FUNCTION_BLOCK GearSequenceGoHome EXTENDS GearSequence IMPLEMENTS ZCore.ISequence
VAR
  _step : ZCore.Step(GearStep.GohomeBegin, GearStep.GohomeEnd);
  _timer : ZAux.Timer;
END_VAR

IF NOT Busy THEN
  RETURN;
END_IF

IF OnStart(_step) THEN
  ; // init custom sequence variables here ...
END_IF

IF OnStop() THEN
  RETURN; // external stop was triggered
END_IF

IF OnHalt() THEN
  ; // Halting := TRUE; // Uncomment to acknowledge that the sequence is halting
END_IF

REPEAT
  LogStep();

  CASE _step.Index OF
    (* -------------------------------------------------------------------------------------------------------------------------------- *)
    GearStep.GoHomeBegin:
    (* -------------------------------------------------------------------------------------------------------------------------------- *)

      _step.SetNext(index:=GearStep.GoHomePositionX);

	(* -------------------------------------------------------------------------------------------------------------------------------- *)
    GearStep.GoHomePositionX:
    (* -------------------------------------------------------------------------------------------------------------------------------- *)
      IF _step.OnEntry()
      THEN        
        _axis.PositionX.MoveAbsoluteAsync(THIS^, _data.Machine.HomePositionX, _data.Machine.SlowspeedX);
      END_IF
      
      Await(obj1:=_axis.PositionX, nextStep:=GearStep.GoHomeRotationC);

	(* -------------------------------------------------------------------------------------------------------------------------------- *)
    GearStep.GoHomeRotationC:
    (* -------------------------------------------------------------------------------------------------------------------------------- *)
      IF _step.OnEntry()
      THEN        
        _axis.RotationC.MoveAbsoluteAsync(THIS^,
            _axis.RotationC.ActualPosition - _parent.PhaseOffsetC + _data.Machine.ToothAngle, _data.Machine.SlowspeedC);
      END_IF
      
      Await(obj1:=_axis.PositionX, nextStep:=GearStep.GoHomeEnd);

    (* -------------------------------------------------------------------------------------------------------------------------------- *)
    GearStep.GoHomeEnd:
    (* -------------------------------------------------------------------------------------------------------------------------------- *)
      SetBusy(FALSE);
  
  ELSE
    Abort('sequence contains unhandled step');
  END_CASE
UNTIL _step.IsNotRepeatable() OR_ELSE NOT Busy END_REPEAT

END_FUNCTION_BLOCK

(* stored: Version 1.1.0.1
   POU GearSequenceGoHome: Id {628f2010-8039-4b2e-b2f4-cdb836ef1b67}, SpecialFunc None *)
